INTERFACE I_Cylinder

PROPERTY delayTimeAfterReachedHP : TIME
GET
END_GET
SET
END_SET
END_PROPERTY

PROPERTY delayTimeAfterReachedWP : TIME
GET
END_GET
SET
END_SET
END_PROPERTY

METHOD fill
VAR_INPUT
END_VAR
END_METHOD

PROPERTY PUBLIC inHP : BOOL
GET
END_GET
END_PROPERTY

PROPERTY interlockMessageHP : STRING(255)
GET
END_GET
END_PROPERTY

PROPERTY interlockMessageWP : STRING(255)
GET
END_GET
END_PROPERTY

PROPERTY PUBLIC inWP : BOOL
GET
END_GET
END_PROPERTY

PROPERTY monitorMovementTimeout : BOOL
GET
END_GET
SET
END_SET
END_PROPERTY

PROPERTY monitorSensorsOverlap : BOOL
GET
END_GET
SET
END_SET
END_PROPERTY

PROPERTY movementTimeout : TIME
GET
END_GET
SET
END_SET
END_PROPERTY

METHOD PUBLIC moveToHP
VAR_INPUT
	Response		: REFERENCE TO TcNexa_Components_TcProcess.FB_MethodResponse;
END_VAR
END_METHOD

METHOD PUBLIC moveToWP
VAR_INPUT
	Response		: REFERENCE TO TcNexa_Components_TcProcess.FB_MethodResponse;
END_VAR
END_METHOD

PROPERTY notUsedSensorHP : BOOL
GET
END_GET
SET
END_SET
END_PROPERTY

PROPERTY notUsedSensorWP : BOOL
GET
END_GET
SET
END_SET
END_PROPERTY

METHOD PUBLIC off
VAR_INPUT
END_VAR
END_METHOD

PROPERTY sensorsOverlapTimeout : TIME
GET
END_GET
SET
END_SET
END_PROPERTY

END_INTERFACE

(* stored: Version 1.1.0.1, ProductVersion 3.1.4024.12
   Itf I_Cylinder: Id {1d011b56-0512-0942-24a1-6da9282bd9a9}
   Folder Property: Id {267c47a5-ae14-0388-13f1-6002b9189ef5}
   Property delayTimeAfterReachedHP: Id {fc60306e-1d25-07b8-2f41-0c1155cb85e4}
   Get Get: Id {d28d7299-deb5-02c3-3ed8-bb02a69fbd6e}
   Set Set: Id {4b4c3fc8-0b1b-0f3e-006e-2945b0b2f22f}
   Property delayTimeAfterReachedWP: Id {560c36ae-0336-0561-08e9-c13567076cd1}
   Get Get: Id {3ccaa96f-e995-09c3-2608-191c276798e7}
   Set Set: Id {5c725605-e158-0463-0450-a679cbe14478}
   Method fill: Id {33ec8077-617b-0751-14af-9288b39bc749}
   Property inHP: Id {7fc6b109-4c17-0f74-1f91-bfe772771f6e}
   Get Get: Id {0febcec0-fe13-095e-389b-1bf0ba6d9f3a}
   Property interlockMessageHP: Id {f1d186f1-b347-0479-1de5-1d214db53257}
   Get Get: Id {583d434f-99e0-07a3-2727-6cf32db4820e}
   Property interlockMessageWP: Id {97b17812-fe17-070a-3397-df80c1df348b}
   Get Get: Id {65976726-eaf2-0b05-0dae-db38e80b7ebd}
   Property inWP: Id {f04e20b6-a035-0f73-1ea1-4d109a16da95}
   Get Get: Id {afbd79aa-1f23-0eb3-04a4-731c69d80fac}
   Property monitorMovementTimeout: Id {92445ae7-5795-0235-10cf-7a358e2fa8fa}
   Get Get: Id {83cf16ba-34a9-089c-38d0-2dec6946bac5}
   Set Set: Id {9212759e-2d20-083b-3f10-8f9568dca510}
   Property monitorSensorsOverlap: Id {39430df8-b8fb-0a57-3acc-d754d3dbca92}
   Get Get: Id {6fad0bab-fae5-0ed2-1302-7cf37c678764}
   Set Set: Id {daf9efc5-33f9-0c16-275b-0f8f39af406b}
   Property movementTimeout: Id {e16a4c43-507d-097a-13c0-bfa35ae5658c}
   Get Get: Id {9f11280f-9700-080e-194f-91813fb1b852}
   Set Set: Id {eb2a27bb-64af-022f-295b-75092f78eb9f}
   Method moveToHP: Id {501d1b69-466f-0a60-3f90-253aff92e997}
   Method moveToWP: Id {ac71704b-c5bc-020b-0be3-2a388b45c2ba}
   Property notUsedSensorHP: Id {a83fc0f9-036f-0f7f-2139-ba83b6b7c306}
   Get Get: Id {c7827522-242e-00b9-20f6-3d3426ad9e01}
   Set Set: Id {ec13cece-a5de-01da-2de8-090ec3d0e38a}
   Property notUsedSensorWP: Id {fb0bcea5-5d93-0321-32eb-5e25af79388e}
   Get Get: Id {13e3f472-9b88-0727-175a-c40f7d6e423f}
   Set Set: Id {28a8aa1e-8fe8-0628-04eb-07f28396b057}
   Method off: Id {11592de3-b27a-0ee4-1cd7-8a6e98a648bd}
   Property sensorsOverlapTimeout: Id {40e1caec-57d4-026c-28c4-d33a2a4ad75f}
   Get Get: Id {af68bc77-08c7-0721-2ab6-0f19ec293e34}
   Set Set: Id {e5d5a6b7-075a-0eb2-3929-b03957f394d1} *)
